(* PLC project actuator, TNI-Software ControlBuild 4.00.17 *)
(* stored: creationDateTime 2005-06-20T11:52:51-01:00 *)

FUNCTION_BLOCK cmd_equipment_library.actuator
  VAR_INPUT  (* CB.group=Modes CB.kind=inputVars *)
    autoMode : BOOL := false;  (* CB.mnemonicPatternPropertyName=<SY>_AUTO_<NU> CB.libelle=Automatic mode *)
    manualMode : BOOL := false;  (* CB.mnemonicPatternPropertyName=<SY>_MANU_<NU> CB.libelle=Manual mode *)
  END_VAR
  VAR_INPUT  (* CB.group=Commands CB.kind=inputVars *)
    autoFwdCmd : BOOL := false;  (* CB.mnemonicPatternPropertyName=<SY>_CMDAVAUTO_<NU> CB.libelle=Automatic forward command *)
    autoBwdCmd : BOOL := false;  (* CB.mnemonicPatternPropertyName=<SY>_CMDARAUTO_<NU> CB.libelle=Automatic backward command *)
    autoHSCmd : BOOL := false;  (* CB.mnemonicPatternPropertyName=<SY>_CMDGVAUTO_<NU> CB.libelle=Automatic high speed command *)
    autoLSCmd : BOOL := false;  (* CB.mnemonicPatternPropertyName=<SY>_CMDPVAUTO_<NU> CB.libelle=Automatic low speed command *)
  END_VAR
  VAR_INPUT  (* CB.group=PushButtons CB.kind=inputVars *)
    forwardPB : BOOL := false;  (* CB.mnemonicPatternPropertyName=<SY>_BPAV_<NU> CB.libelle=Forward pushbutton *)
    backwardPB : BOOL := false;  (* CB.mnemonicPatternPropertyName=<SY>_BPAR_<NU> CB.libelle=Backward pushbutton *)
    highSpeedPB : BOOL := false;  (* CB.mnemonicPatternPropertyName=<SY>_BPGV_<NU> CB.libelle=High speed pushbutton *)
    lowSpeedPB : BOOL := false;  (* CB.mnemonicPatternPropertyName=<SY>_BPPV_<NU> CB.libelle=Low speed pushbutton *)
    stopPB : BOOL := false;  (* CB.mnemonicPatternPropertyName=<SY>_BPARRET_<NU> CB.libelle=Stop pushbutton *)
  END_VAR
  VAR_INPUT  (* CB.kind=inputVars *)
    generalFault : BOOL := false;  (* CB.mnemonicPatternPropertyName=<SY>_DEF_<NU> CB.libelle=General fault of the engine *)
  END_VAR
  VAR_OUTPUT  (* CB.group=Orders CB.kind=outputVars *)
    forwardCmd : BOOL := false;  (* CB.mnemonicPatternPropertyName=fwdCmd<SY><NU> CB.libelle=Forward command *)
    backwardCmd : BOOL := false;  (* CB.mnemonicPatternPropertyName=bwdCmd<SY><NU> CB.libelle=Backward command *)
    highSpeedCmd : BOOL := false;  (* CB.mnemonicPatternPropertyName=hSCmd<SY><NU> CB.libelle=High speed command *)
    lowSpeedCmd : BOOL := false;  (* CB.mnemonicPatternPropertyName=lSCmd<SY><NU> CB.libelle=Low speed command *)
  END_VAR

(* LD diagram, written out as Structured Text *)
1:
forwardCmd := (autoMode AND autoFwdCmd OR manualMode AND (forwardCmd OR forwardPB AND NOT backwardPB) AND NOT stopPB AND NOT backwardCmd) AND NOT generalFault;
2:
backwardCmd := (autoMode AND autoBwdCmd OR manualMode AND (backwardCmd OR backwardPB AND NOT forwardPB) AND NOT stopPB AND NOT forwardCmd) AND NOT generalFault;
3:
highSpeedCmd := (autoMode AND autoHSCmd OR manualMode AND (highSpeedPB OR highSpeedCmd) AND NOT lowSpeedPB) AND NOT generalFault;
lowSpeedCmd := (autoMode AND autoLSCmd OR manualMode AND (lowSpeedPB OR lowSpeedCmd) AND NOT highSpeedPB) AND NOT generalFault;
END_FUNCTION_BLOCK
